(* IEC 61131-3 sources: mastertool-rankine-bridge/tests/fixtures/sample_gvls, 1 file *)

(* ---- GVL_Simples.st ---- *)
(* GVL sintetica para testes de parser *)
VAR_GLOBAL CONSTANT
    MAX_EIXOS : INT := 4;
END_VAR
VAR_GLOBAL
    xEmergencia : BOOL;
    arEixos     : ARRAY[1..MAX_EIXOS] OF REAL;
END_VAR
